// TIA Portal V20 export
FUNCTION_BLOCK "FB_Powermeter"   // FB433, SCL
{ S7_Optimized_Access := 'TRUE' }
// stored: AutoNumber false, MemoryReserve 100, SetENOAutomatically false
   VAR
      sPowerMeterWorkPos : Bool;
      sPowerMeterHomePos : Bool;
      sPowerMeterToWorkMoveReq : Bool;
      sPowerMeterToHomeMoveReq : Bool;
      sPowerMeterJogMode : Bool;
      sPowermeterCylinder : "FB_CmdCylinder";
      sPowermeterInHomePos { S7_SetPoint := 'True'} : Bool;
      sPowermeterInMiddlePos : Bool;
      sPowermeterInWorkPos : Bool;
      sPowerMeterCylErrorCode : Int;
      sPowerMeterHomePosCtrlTimer : TON_TIME;
      sPowerMeterWorkPosCtrlTimer : TON_TIME;
      sMeasurePowerLaser { S7_SetPoint := 'True'} : Bool;
      sRTLaserMeasureON : R_TRIG;
      sLaserPowerValue { S7_SetPoint := 'True'} : Real;
      sWeightFactor : Real;
      sAlpha : Real;
      sDateAndTime : DTL;
      sActualMeasPower : Real;
      sTolMin : Real;
      sTolMax : Real;
      sResetMeasures : Bool;
      sPowerMeterSeq : "FB_PowerMeterSeq";
      RT_StartArchive { S7_SetPoint := 'True'} : R_TRIG;
      sArchivePmValues { S7_SetPoint := 'True'} : Array[0..4] of Real;
   END_VAR
   VAR_TEMP
      tAxis01_X1SafePos : Bool;
      tLaserMeasureON : Bool;
      tActualMeasure : Int;
      tRetVal : Int;
      tAverageValue : Real;
      tStandardDeviation : Real;
      tTempReal : Real;
      tIndex : Int;
   END_VAR
   VAR CONSTANT
      POWERMETER_HOME_POS_CTRL_TIME : Time := T#6s;
      POWERMETER_WORK_POS_CTRL_TIME : Time := T#6s;
   END_VAR
BEGIN
   REGION Description header 
       //==================================================================================
       // POSALUX Swiss SA / (C) Copyright 2025
       //----------------------------------------------------------------------------------
       // Title: Initialization of axis
       // Comment/Function: 
       // Author: Fabien WALDT
       // Engineering: TIA Portal v17
       //----------------------------------------------------------------------------------
       // Change log table:
       // Version  | Date     | Expert in charge | Changes applied
       // ---------|----------|------------------|-----------------------------------------
       // 00.00.01 | 20250501 | WFA              | First released version
       // =================================================================================
   END_REGION

   REGION Axis01_X on safe position
      // Check position Axis01_X to release the powermeter
       #tAxis01_X1SafePos := "DB_AxisPosition".sAxis01_X."$AA_IM" >= "DB_AxisPosition".sAxis01_X."$MA_POS_LIMIT_PLUS" - 10.0;
   END_REGION

   REGION Blocking Axis01_X
       // Blocking Axis01_X if Powermeter is in measuring position
       "LBP_Axis01_X".A_ASpDisable := NOT #sPowerMeterHomePos OR #sPowerMeterWorkPos; 
   END_REGION
   REGION PowerMeter Sequence
       // #sPowerMeterSeq(iStartSeqCond:=#sPowerMeterSeq.iStartSeqCond,
       //                 iJobReq:=#sPowerMeterSeq.iJobReq,
       //                 iPowerMeterHomePos:=#sPowerMeterSeq.iPowerMeterHomePos,
       //                 iPowerMeterWorkPos:=#sPowerMeterSeq.iPowerMeterWorkPos,
       //                 iNC_Stopped:=#sPowerMeterSeq.iNC_Stopped,
       //                 iPLC_DateAndTime:="DB_ReadDateAndTime".sDateAndTime,
       //                 iStepPause:=#sPowerMeterSeq.iStepPause,
       //                 rMinValue:=#sPowerMeterSeq.rMinValue,
       //                 rMaxValue:=#sPowerMeterSeq.rMaxValue,
       //                 iStopOption:=#sPowerMeterSeq.iStopOption,
       //                 rMeasureValue:=#sPowerMeterSeq.rMeasureValue,
       //                 iMeasureDone:=#sPowerMeterSeq.iMeasureDone,
       //                 oPowerMetertoHomeReq=>#sPowerMeterSeq.oPowerMetertoHomeReq,
       //                 oPowerMetertoWorkReq=>#sPowerMeterSeq.oPowerMetertoWorkReq,
       //                 oStopNC_Req=>#sPowerMeterSeq.oStopNC_Req,
       //                 oMsgBadMeasure=>#sPowerMeterSeq.oMsgBadMeasure,
       //                 oStartMeasure=>#sPowerMeterSeq.oStartMeasure,
       //                 oStartArchive=>#sPowerMeterSeq.oStartArchive,
       //                 oRID=>#sPowerMeterSeq.oRID);
   END_REGION

   REGION Powermeter Key / LED Management
       // Disable Powemeter Key[1] if not Jog Mode
       "DB_McpKeyboardSignals".sK1_Powermeter.sKeyDisable := NOT "LBP_ModeGroup".E_JOG OR NOT #tAxis01_X1SafePos OR "DB_GestionWorkingModes".sMCP_KxxKeysDisable;
       "DB_HmiKeyboardSignals".sK1_Powermeter.sKeyDisable := NOT "LBP_ModeGroup".E_JOG OR NOT #tAxis01_X1SafePos;

       // Set/Reset Toggle Powemeter Key[1]
       IF #sPowerMeterSeq.oPowerMetertoWorkReq THEN    // Powermeter to work position
           "DB_McpKeyboardSignals".sK1_Powermeter.sKeySWToggleStatus := TRUE;
           "DB_HmiKeyboardSignals".sK1_Powermeter.sKeySWToggleStatus := TRUE;
       END_IF;
       IF #sPowerMeterSeq.oPowerMetertoHomeReq OR     // Powermeter to home position
           "LBP_Chan1".A_Reset  THEN
           "DB_McpKeyboardSignals".sK1_Powermeter.sKeySWToggleStatus := FALSE;
           "DB_HmiKeyboardSignals".sK1_Powermeter.sKeySWToggleStatus := FALSE;
           END_IF;

       // Powemeter LED[1] Animation
           "DB_McpKeyboardSignals".sK1_Powermeter.sLedSWStatus :=
           ("DB_McpKeyboardSignals".sK1_Powermeter.sKeySWToggleStatus AND #tAxis01_X1SafePos)
           OR ("DB_McpKeyboardSignals".sK1_Powermeter.sKeySWToggleStatus AND "Clock_2Hz");

           "DB_HmiKeyboardSignals".sK1_Powermeter.sLedSWStatus :=
           ("DB_HmiKeyboardSignals".sK1_Powermeter.sKeySWToggleStatus AND #tAxis01_X1SafePos)
           OR ("DB_HmiKeyboardSignals".sK1_Powermeter.sKeySWToggleStatus AND "Clock_2Hz");
   END_REGION

   REGION Powermeter in work position move request
       #sPowerMeterToWorkMoveReq :=
       ("DB_McpKeyboardSignals".sK1_Powermeter.sKeySWToggleStatus AND NOT "MCP1_In".incVar)
       OR ("DB_HmiKeyboardSignals".sK1_Powermeter.sKeySWToggleStatus AND NOT "MCP1_In".incVar)
       AND #tAxis01_X1SafePos;
   END_REGION

   REGION Powermeter in home position move request
       #sPowerMeterToHomeMoveReq :=
       (NOT "DB_McpKeyboardSignals".sK1_Powermeter.sKeySWToggleStatus AND
        NOT "DB_HmiKeyboardSignals".sK1_Powermeter.sKeySWToggleStatus);
   END_REGION

   REGION Powermeter in JOG Mode
       #sPowerMeterJogMode := "LBP_ModeGroup".E_JOG AND "MCP1_Out".LEDincVar;
   END_REGION

   REGION Move/Control Powermeter Cylinder
       #sPowermeterCylinder(iEMinus:="DB_DigitalInputs".sPowerMeterBackCtrl.sSWStatus,
                            iEPlus:="DB_DigitalInputs".sPowerMeterFrontCtrl.sSWStatus,
                            iMinusCmd:=#sPowerMeterToHomeMoveReq,
                            iPlusCmd:=#sPowerMeterToWorkMoveReq,
                            iJOGCmd:=#sPowerMeterJogMode,
                            iMonitorTime:=T#8s,
                            ioQMinus:="DB_DigitalOutputs".sPowerMeterRetract.sSWStatus,
                            ioQPlus:="DB_DigitalOutputs".sPowerMeterAdvance.sSWStatus,
                            oMinusPos=>#sPowermeterInHomePos,
                            oMiddlePos=>#sPowermeterInMiddlePos,
                            oPlusPos=>#sPowermeterInWorkPos,
                            oErrorCode=>#sPowerMeterCylErrorCode);
   END_REGION

   REGION Powermeter Cylinder Positions
       #sPowerMeterHomePos := #sPowermeterCylinder.iEMinus;
       #sPowerMeterWorkPos := #sPowermeterCylinder.iEPlus;
   END_REGION

   REGION Powermeter Cylinder Alarms
       "LBP_AlarmMsgs".UserA[6].A70UUxx[62] := #sPowerMeterCylErrorCode = 1;    // Msg: 700662 "Alarm power meter entry"
       "LBP_AlarmMsgs".UserA[6].A70UUxx[63] := #sPowerMeterCylErrorCode = 2;    // Msg: 700663 "Alarm power meter exit"
   END_REGION

   REGION Monitoring Cylinder in home position
       #sPowerMeterHomePosCtrlTimer(IN:=#sPowerMeterToHomeMoveReq AND NOT #sPowermeterInHomePos,
                                    PT:=#POWERMETER_HOME_POS_CTRL_TIME);

       IF #sPowerMeterHomePosCtrlTimer.Q THEN
           "LBP_AlarmMsgs".ChanA[1].FDD_5C00xx[0] := TRUE;     // Msg: 510000 "Power meter runtimeerror workposition"
       END_IF;

       IF "LBP_Chan1".A_Reset THEN
           "LBP_AlarmMsgs".ChanA[1].FDD_5C00xx[0] := FALSE;    // Msg: 510000 "Power meter runtimeerror workposition"
       END_IF;

       // Read-in disable during movement
       IF #sPowerMeterToHomeMoveReq AND NOT #sPowermeterInHomePos THEN
           "LBP_AlarmMsgs".Chan[1].RID[6] := TRUE;
       END_IF;

       IF #sPowermeterInHomePos OR "LBP_Chan1".A_Reset THEN
           "LBP_AlarmMsgs".Chan[1].RID[6] := FALSE;            
       END_IF;
   END_REGION

   REGION Monitoring Cylinder in work position
       #sPowerMeterWorkPosCtrlTimer(IN := #sPowerMeterToWorkMoveReq AND NOT #sPowermeterInWorkPos,
                                    PT := #POWERMETER_WORK_POS_CTRL_TIME);

       IF #sPowerMeterWorkPosCtrlTimer.Q THEN
           "LBP_AlarmMsgs".ChanA[1].FDD_5C00xx[0] := TRUE;     // Msg: 510000 "Power meter runtimeerror workposition"
       END_IF;

       IF "LBP_Chan1".A_Reset THEN
           "LBP_AlarmMsgs".ChanA[1].FDD_5C00xx[0] := FALSE;    // Msg: 510000 "Power meter runtimeerror workposition"
       END_IF;

       // Read-in disable during movement
       IF #sPowerMeterToWorkMoveReq AND NOT #sPowermeterInWorkPos THEN
           "LBP_AlarmMsgs".Chan[1].RID[7] := TRUE;
       END_IF;

       IF #sPowermeterInWorkPos OR "LBP_Chan1".A_Reset THEN
           "LBP_AlarmMsgs".Chan[1].RID[7] := FALSE;            
       END_IF;
   END_REGION

   REGION Start/Stop measure laser power   
       // M21: Start measure laser power
       IF #sPowerMeterSeq.oStartMeasure THEN
           #sMeasurePowerLaser := TRUE;
       END_IF;

       // M22: Stop measure laser power
       IF NOT #sPowerMeterSeq.oStartMeasure OR "MCP1_In".reset THEN
           #sMeasurePowerLaser := FALSE;
       END_IF;
   END_REGION

   REGION Power value calculation  
       #tLaserMeasureON := #sMeasurePowerLaser OR #sPowerMeterJogMode;

       // Init Powermeter value when restart
       #sRTLaserMeasureON(CLK:=#tLaserMeasureON AND #sPowermeterInWorkPos);
       IF #sRTLaserMeasureON.Q THEN
           #sLaserPowerValue := 0.0;
       END_IF;

       // Power value calculation
       IF #tLaserMeasureON AND #sPowermeterInWorkPos THEN
           #sLaserPowerValue := #sAlpha * "DB_AnalogInputs".sLaserPowerMeter.sSWRealValue +
           (1 - #sAlpha) * #sLaserPowerValue;
           "LBP_NC".A_Setval_anaIn3 := DINT_TO_WORD(REAL_TO_DINT(#sLaserPowerValue * #sWeightFactor));
           "LBP_NC".A_InMask_anaIn3 := TRUE;
       END_IF;
   END_REGION

   REGION Archive 5 last values
       #RT_StartArchive(CLK := #sPowerMeterSeq.oStartArchive);

       IF #RT_StartArchive.Q THEN
           FOR #tIndex := 1 TO 4 DO
               #sArchivePmValues[#tIndex] := #sArchivePmValues[#tIndex - 1];
           END_FOR;
           #sArchivePmValues[0] := #sLaserPowerValue;
       END_IF;
   END_REGION

   REGION Date et Time reading
       #tRetVal := RD_SYS_T(OUT => #sDateAndTime);
   END_REGION

   REGION Measurement archiving
       IF "LBP_Chan1".MDyn[39] THEN
           #tActualMeasure := "DB_PowermeterMeasures".ActualMeasure + 1;
           IF #tActualMeasure >= "DB_PowermeterMeasures".NbMeasure THEN
               #tActualMeasure := 0;
               "DB_PowermeterMeasures".Table_full := TRUE;  // WFA Bit jamais remis à 0
           END_IF;

           "DB_PowermeterMeasures".Measures[#tActualMeasure].Day_meas := DTL_TO_DATE(#sDateAndTime);
           "DB_PowermeterMeasures".Measures[#tActualMeasure].Time_day := DTL_TO_TOD(#sDateAndTime);

           #sActualMeasPower := "LBP_Chan1".H1;

           "DB_PowermeterMeasures".ActualTotalMeas :=
           #sActualMeasPower
           - "DB_PowermeterMeasures".Measures[#tActualMeasure].ValuePower
           + "DB_PowermeterMeasures".ActualTotalMeas;

           "DB_PowermeterMeasures".Measures[#tActualMeasure].ValuePower := #sActualMeasPower;

           REGION Average and Standard Deviation Calculation
               IF "DB_PowermeterMeasures".Table_full THEN
                   #tActualMeasure := 100;
               ELSIF #tActualMeasure < 0 THEN
                   #tActualMeasure := 1;
               END_IF;

               #tAverageValue := "DB_PowermeterMeasures".ActualTotalMeas / #tActualMeasure;

               #tTempReal := ((#tAverageValue * -2.0 * "DB_PowermeterMeasures".ActualTotalMeas) / #tActualMeasure) + #tAverageValue;

               #tStandardDeviation := SQRT(("DB_PowermeterMeasures".ActualMeasure * "DB_PowermeterMeasures".ActualMeasure / #tActualMeasure) + #tTempReal);
           END_REGION

           REGION Compute CM  (" Tol+" - " Tol-" ) / (6 Sigma) process capability index
               IF #tStandardDeviation * 6.0 > 0.0001 THEN
                   #tTempReal := #tStandardDeviation;
               ELSE
                   #tTempReal := 1.0;
               END_IF;

               "DB_PowermeterMeasures".Measures[#tActualMeasure].ValueCM :=
               (#sTolMax - #sTolMin) / #tTempReal;

               "DB_PowermeterMeasures".ActualMeasure := #tActualMeasure;
           END_REGION
       END_IF;
   END_REGION

   REGION Reset Measures
       IF #sResetMeasures THEN
           FOR #tIndex := 0 TO "DB_PowermeterMeasures".NbMeasure - 1 DO
               "DB_PowermeterMeasures".Measures[#tIndex].Job_meas := -1;
               "DB_PowermeterMeasures".Measures[#tIndex].ValuePower := 0.0;
               "DB_PowermeterMeasures".Measures[#tIndex].ValueCM := 0.0;
           END_FOR;
       END_IF;
   END_REGION
END_FUNCTION_BLOCK
